TYPE ST_MESSAGE_STATE :
STRUCT
  State         : E_MESSAGE_STATE;  // as always... combined value of Cmd equivalent and e_progress
END_STRUCT
END_TYPE

(* stored: Version 1.1.0.1
   DUT ST_MESSAGE_STATE: Id {b62350f3-8716-4d9c-9505-456f0834ca41} *)
